SUBAPPLICATION Ventilsteuerung_Uebung_017 (* Control Audio Signal *)
  (* Standard: 61499-2 *)
  (* Version 1.0, 2023-10-23, franz *)
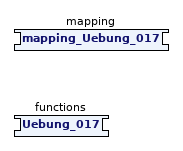
  SUBAPPS
    mapping : mapping_Uebung_017;
    functions : Uebung_017;
  END_SUBAPPS
END_SUBAPPLICATION
